KUKA KRL program: e_fraes1.src, e_fraes1.dat

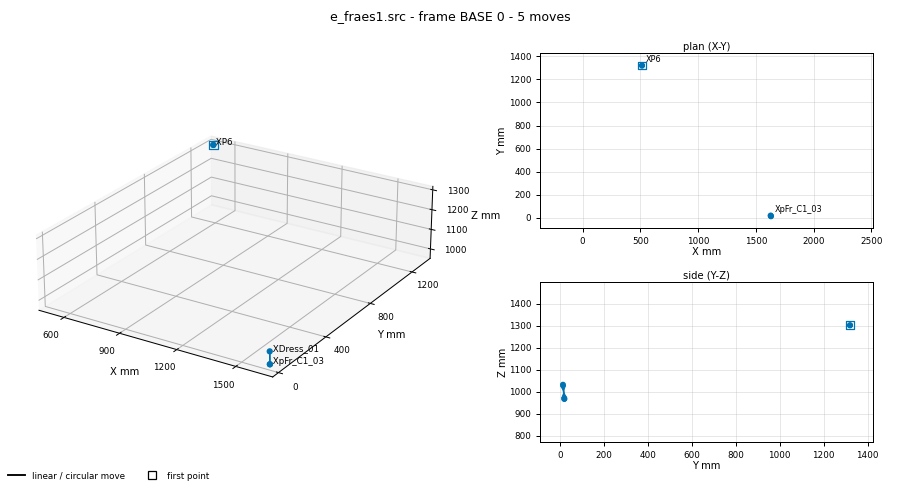
[picture p0: tool path of e_fraes1.src in frame BASE 0, 5 of 7 moves have a stored position in this frame; points joined in program order, loops and branches not executed]
--- e_fraes1.src ---
&ACCESS RVP3
&REL 172
&COMMENT Fresa C1
&PARAM DISKPATH = KRC:\R1\Program\SERVICE
&PARAM TEMPLATE = C:\KRC\Roboter\Template\vorgabe
&PARAM EDITMASK = *
DEF e_Fraes1( )
;FOLD INI
  ;FOLD BASISTECH INI
    GLOBAL INTERRUPT DECL 3 WHEN $STOPMESS==TRUE DO IR_STOPM ( )
    INTERRUPT ON 3
    BAS (#INITMOV,0 )
  ;ENDFOLD (BASISTECH INI)
;FOLD SPOTTECH INI
USERSPOT(#INIT)
;ENDFOLD (SPOTTECH INI)
;FOLD GRIPPERTECH INI
USER_GRP(0,DUMMY,DUMMY,GDEFAULT)
;ENDFOLD (GRIPPERTECH INI)
  ;FOLD USER INI
    ;Make your modifications here

  ;ENDFOLD (USER INI)
;ENDFOLD (INI)

; Caracterização dos meios de produção:
; Versão Atual:
; 15/07/2013 12:00 Name: P13.050-R4 CHANGES: Fresa
; C1


chk_w1_wechs_ok ( )     ; CHECK FERRAMENTA: C1


;FOLD PTP P6 Vel=100 % PDAT0 Tool[1]:GUN_C1 Base[0];%{PE}%R 8.2.20,%MKUKATPBASIS,%CMOVE,%VPTP,%P 1:PTP, 2:P6, 3:, 5:100, 7:PDAT0
$BWDSTART=FALSE
PDAT_ACT=PPDAT0
FDAT_ACT=FP6
BAS(#PTP_PARAMS,100)
PTP XP6
;ENDFOLD
;FOLD PTP P3 CONT Vel=100 % PDAT15 Tool[1]:GUN_C1 Base[0];%{PE}%R 8.2.20,%MKUKATPBASIS,%CMOVE,%VPTP,%P 1:PTP, 2:P3, 3:C_DIS, 5:100, 7:PDAT15
$BWDSTART=FALSE
PDAT_ACT=PPDAT15
FDAT_ACT=FP3
BAS(#PTP_PARAMS,100)
PTP XP3 C_DIS
;ENDFOLD
;FOLD PTP pFr_C1_03 CONT Vel=100 % PDAT18 Tool[1]:GUN_C1 Base[0];%{PE}%R 8.2.20,%MKUKATPBASIS,%CMOVE,%VPTP,%P 1:PTP, 2:pFr_C1_03, 3:C_DIS, 5:100, 7:PDAT18
$BWDSTART=FALSE
PDAT_ACT=PPDAT18
FDAT_ACT=FpFr_C1_03
BAS(#PTP_PARAMS,100)
PTP XpFr_C1_03 C_DIS
;ENDFOLD

;FOLD ; PONTO DE FRESAGEM;%{PE}%R 8.2.20,%MKUKATPBASIS,%CCOMMENT,%VNORMAL,%P 2:PONTO  DE  FRESAGEM
;ENDFOLD
;FOLD TIP.LIN_ Dress_01, Spot Gun 1 , RETR open , Tool[1], Base[0], EXT.TCP=FALSE;%{PE}%MKUKATPUSER
FDAT_ACT=FDress_01
BAS(#FRAMES)
LIN  XDress_01
S_ACT.GUN=1
S_ACT.RETR=#opn
S_READY=FALSE
USERSPOT (#DRESS,S_ACT )
WAIT FOR  S_READY
;ENDFOLD

;FOLD LIN pFr_C1_05 CONT Vel=0.25 m/s CPDAT3 Tool[1]:GUN_C1 Base[0];%{PE}%R 8.2.20,%MKUKATPBASIS,%CMOVE,%VLIN,%P 1:LIN, 2:pFr_C1_05, 3:C_DIS C_DIS, 5:0.25, 7:CPDAT3
$BWDSTART=FALSE
LDAT_ACT=LCPDAT3
FDAT_ACT=FpFr_C1_05
BAS(#CP_PARAMS,0.25)
LIN XpFr_C1_05 C_DIS C_DIS
;ENDFOLD

;FOLD PTP pFr_C2_09 PDAT6 SPOT Gun=1 RETR OPN PgNo1=251 ACTIVE=1 Tool[1]:GUN_C1 Base[1]:ACTROS;%{PE}%R 8.2.2,%MKUKATPSPOT,%CSPOT,%VPTP,%P 1:PTP, 2:pFr_C2_09, 3:, 5:100, 7:PDAT6, 10:1, 12:#FIRST, 14:#OPN, 16:251, 18:1, 20:0, 22:0, 24:1, 25:NORMAL
$BWDSTART=FALSE
PDAT_ACT=PPDAT6
FDAT_ACT=FpFr_C2_09
BAS(#PTP_PARAMS,PPDAT6.VEL)
S_ACT.GUN=1
S_ACT.PAIR=SDEFAULT.PAIR
S_ACT.RETR=#OPN
S_ACT.CLO_TM=1
S_ACT.PGNO1=251
S_ACT.PGNO2=SDEFAULT.PGNO2
S_ACT.PRESS1=SDEFAULT.PRESS1
S_ACT.PRESS2=SDEFAULT.PRESS2
S_READY=FALSE
PTP XpFr_C2_09
USERSPOT(#SPOT, S_ACT)
WAIT FOR S_READY
;ENDFOLD
;FOLD PTP pFr_C1_07 CONT Vel=100 % PDAT4 Tool[1]:GUN_C1 Base[0];%{PE}%R 8.2.20,%MKUKATPBASIS,%CMOVE,%VPTP,%P 1:PTP, 2:pFr_C1_07, 3:C_DIS, 5:100, 7:PDAT4
$BWDSTART=FALSE
PDAT_ACT=PPDAT4
FDAT_ACT=FpFr_C1_07
BAS(#PTP_PARAMS,100)
PTP XpFr_C1_07 C_DIS
;ENDFOLD

END

--- e_fraes1.dat ---
&ACCESS RVP3
&REL 172
&COMMENT Fresa C1
&PARAM DISKPATH = KRC:\R1\Program\SERVICE
&PARAM TEMPLATE = C:\KRC\Roboter\Template\vorgabe
&PARAM EDITMASK = *
DEFDAT  e_fraes1
;FOLD EXTERNAL DECLARATIONS;%{PE}%MKUKATPBASIS,%CEXT,%VCOMMON,%P
;FOLD GRIPPERTECH EXT
EXT  H50 (INT  :IN,INT  :IN,INT  :IN,GRP_TYP  :IN )
;ENDFOLD (GRIPPERTECH EXT)
;FOLD SPOTTECH EXT
EXT  USERSPOT (S_COMMAND  :IN,SPOT_TYPE  :IN )
;ENDFOLD (SPOTTECH EXT)
;FOLD BASISTECH EXT;%{PE}%MKUKATPBASIS,%CEXT,%VEXT,%P
EXT  BAS (BAS_COMMAND  :IN,REAL  :IN )
DECL INT SUCCESS
;ENDFOLD (BASISTECH EXT)
;FOLD USER EXT;%{E}%MKUKATPUSER,%CEXT,%VEXT,%P
;Make your modifications here

;ENDFOLD (USER EXT)
;ENDFOLD (EXTERNAL DECLARATIONS)
DECL BASIS_SUGG_T LAST_BASIS={POINT1[] "P0                      ",POINT2[] "P0                      ",CP_PARAMS[] "CPDAT0                  ",PTP_PARAMS[] "PDAT0                   ",CONT[] "                        ",CP_VEL[] "2.0                     ",PTP_VEL[] "100                     ",SYNC_PARAMS[] "SYNCDAT                 ",SPL_NAME[] "S0                      "}
DECL LDAT LCPDAT3={VEL 2.0,ACC 100.0,APO_DIST 100.0,APO_FAC 50.0,AXIS_VEL 100.0,AXIS_ACC 100.0,ORI_TYP #VAR,CIRC_TYP #BASE,JERK_FAC 50.0,GEAR_JERK 50.0,EXAX_IGN 0}
DECL PDAT PPDAT4={VEL 100.0,ACC 100.0,APO_DIST 25.0,APO_MODE #CDIS}
DECL FDAT FDress_01={TOOL_NO 1,BASE_NO 0,IPO_FRAME #BASE}
DECL E6POS XDress_01={X 1630.65405,Y 14.1011696,Z 1031.448,A -90.6816483,B -0.423877388,C 0.0973087475,S 2,T 3,E1 -351.023407,E2 0.0,E3 0.0,E4 0.0,E5 0.0,E6 0.0}
DECL E6POS XPFR_C1_03={X 1628.16699,Y 20.2751198,Z 966.990723,A -90.7101288,B -0.783713698,C 0.0916769281,S 2,T 3,E1 -353.278198,E2 0.0,E3 0.0,E4 0.0,E5 0.0,E6 0.0}
DECL FDAT FpFr_C1_03={TOOL_NO 1,BASE_NO 0,IPO_FRAME #BASE,POINT2[] " ",TQ_STATE FALSE}
DECL E6POS XpFr_C1_05={X 1628.15503,Y 20.2848492,Z 966.991211,A -90.7113724,B -0.783427119,C 0.0911598131,S 2,T 3,E1 -353.28299,E2 0.0,E3 0.0,E4 0.0,E5 0.0,E6 0.0}
DECL FDAT FpFr_C1_05={TOOL_NO 1,BASE_NO 0,IPO_FRAME #BASE,POINT2[] " ",TQ_STATE FALSE}
DECL E6POS XPFR_C1_07={X 514.272095,Y 1319.72498,Z 1301.66797,A -120.6903,B 9.26167679,C -0.697597504,S 2,T 11,E1 -353.286804,E2 0.0,E3 0.0,E4 0.0,E5 0.0,E6 0.0}
DECL FDAT FpFr_C1_07={TOOL_NO 1,BASE_NO 0,IPO_FRAME #BASE,POINT2[] " ",TQ_STATE FALSE}
DECL SPOT_SUGG_T LAST_SPOT={GUN[] "1                       ",RETR_CMD[] "#CLO                    ",CHOISE[] "#FIRST                  ",CLO_TM[] "1                       ",PGNO1[] "1                       ",PRESS1[] "0                       ",PGNO2[] "1                       ",PRESS2[] "0                       ",SPOT_PARAMS[] "NORMAL                  "}
DECL E6POS XPFR_C2_09={X -7212.84277,Y 3854.78711,Z -433.009491,A 24.3302803,B -0.195081696,C 3.55001903,S 2,T 3,E1 -353.284088,E2 0.0,E3 0.0,E4 0.0,E5 0.0,E6 0.0}
DECL FDAT FpFr_C2_09={TOOL_NO 1,BASE_NO 1,IPO_FRAME #BASE,POINT2[] " ",TQ_STATE FALSE}
DECL PDAT PPDAT6={VEL 100.0,ACC 100.0,APO_DIST 100.0}
DECL E6POS XP3={X -7485.52393,Y 3850.81592,Z -557.766174,A 24.3302498,B -0.195091203,C 3.55002499,S 2,T 3,E1 -353.283997,E2 0.0,E3 0.0,E4 0.0,E5 0.0,E6 0.0}
DECL FDAT FP3={TOOL_NO 2,BASE_NO 2,IPO_FRAME #BASE,POINT2[] " ",TQ_STATE FALSE}
DECL PDAT PPDAT15={VEL 100.0,ACC 100.0,APO_DIST 100.0,APO_MODE #CDIS}
DECL PDAT PPDAT0={VEL 100.0,ACC 100.0,APO_DIST 100.0}
DECL E6POS XP6={X 514.271179,Y 1319.71704,Z 1301.66699,A -120.691002,B 9.26141739,C -0.69756192,S 2,T 11,E1 -353.286499,E2 0.0,E3 0.0,E4 0.0,E5 0.0,E6 0.0}
DECL FDAT FP6={TOOL_NO 1,BASE_NO 0,IPO_FRAME #BASE,POINT2[] " ",TQ_STATE FALSE}
DECL PDAT PPDAT18={VEL 100.0,ACC 100.0,APO_DIST 100.0,APO_MODE #CDIS}
ENDDAT
